TYPE TRunCmdLoader :
	(
		RCLo_None,
		RCLo_TakePart,
		RCLo_GivePart,
		RCLo_TakePlate,
		RCLo_GivePlate,
		RCLo_Cleaning,
		RCLo_PrepareTakePart,
		RCLo_PrepareDropPart,
		RCLo_MoveToSafe,
		RCLo_SwitchPlate,
		RCLo_EndOfRecipe,
		RCLo_ScanPlate
	);
END_TYPE

(* stored: Version 1.1.0.1, ProductVersion 3.1.4022.12
   DUT TRunCmdLoader: Id {244ce1b2-c675-4ff0-8116-8eadfbb43d07} *)
